// Mitsubishi GX Works2 project: TEx01   PLC: Q02/Q02H

PROGRAM MAIN
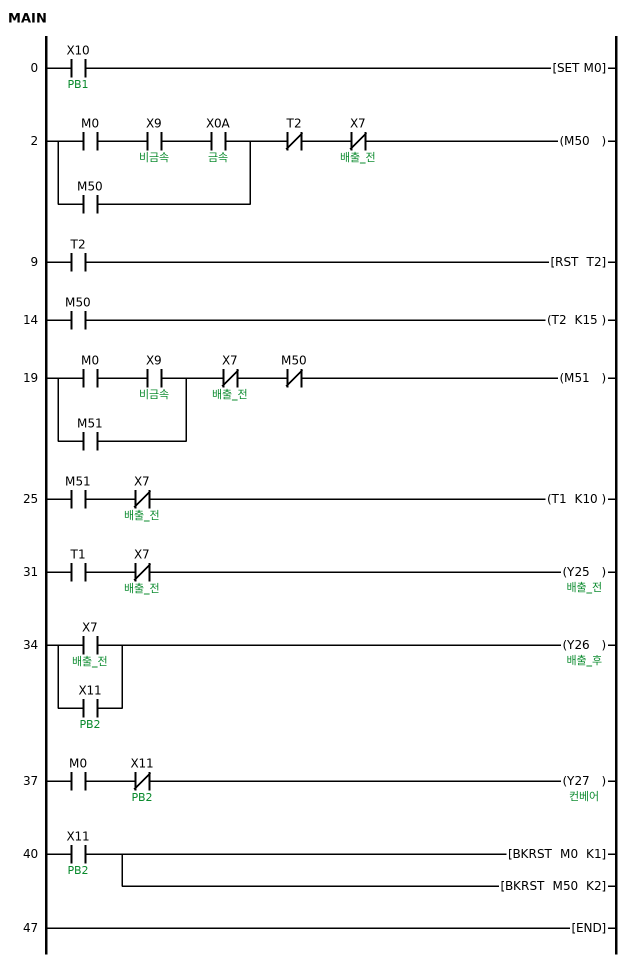
0     LD      X10  ; PB1
      SET     M0
2     LD      M0
      AND     X9  ; 비금속
      AND     X0A  ; 금속
      OR      M50
      ANI     T2
      ANI     X7  ; 배출_전
      OUT     M50
9     LD      T2
      RST     T2
14    LD      M50
      OUT     T2 K15
19    LD      M0
      AND     X9  ; 비금속
      OR      M51
      ANI     X7  ; 배출_전
      ANI     M50
      OUT     M51
25    LD      M51
      ANI     X7  ; 배출_전
      OUT     T1 K10
31    LD      T1
      ANI     X7  ; 배출_전
      OUT     Y25  ; 배출_전
34    LD      X7  ; 배출_전
      OR      X11  ; PB2
      OUT     Y26  ; 배출_후
37    LD      M0
      ANI     X11  ; PB2
      OUT     Y27  ; 컨베어
40    LD      X11  ; PB2
      BKRST   M0 K1
      BKRST   M50 K2
47    END
END_PROGRAM

// device comments not shown above
X0  ; 공급_후
X1  ; 공급_전
X2  ; 드릴_상
X3  ; 드릴_하
X4  ; 송출_후
X5  ; 송출_전
X6  ; 배출_후
X8  ; 매거진
X12  ; PB3
Y20  ; 공급_전
Y21  ; 공급_후
Y22  ; 드릴_하강
Y23  ; 송출_전
Y24  ; 송출_후
Y28  ; 가공드
Y29  ; 적색
Y2A  ; 황색
Y2B  ; 녹색
